TYPE ST_Tray :
STRUCT
	crop_id : INT;
	crop_status : INT;
	level : INT;
	plant_id : INT;
	stack : INT;
	stage : INT;
	plant : ST_PlantConfig;
END_STRUCT
END_TYPE

(* stored: Version 1.1.0.1, ProductVersion 3.1.4024.12
   DUT ST_Tray: Id {4503b853-b3b8-419a-bab1-cfe3b76a9511} *)
